TYPE st_COE_Parameter_Out :
STRUCT
	sName		: STRING(22);
	nWert		: LREAL;

END_STRUCT
END_TYPE

(* stored: Version 1.1.0.1
   DUT st_COE_Parameter_Out: Id {12ae7cba-6d98-4189-b188-342c0147cc93} *)
